FUNCTION_BLOCK INITswitch
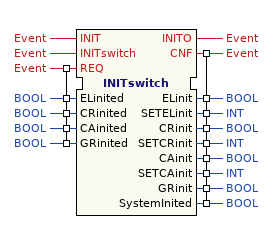
  EVENT_INPUT
    INIT;
    INITswitch;
    REQ WITH ELinited, CRinited, CAinited, GRinited;
  END_EVENT
  EVENT_OUTPUT
    INITO;
    CNF WITH ELinit, SETELinit, CRinit, SETCRinit, CAinit, SETCAinit, GRinit, SystemInited;
  END_EVENT
  VAR_INPUT
    ELinited : BOOL;
    CRinited : BOOL;
    CAinited : BOOL;
    GRinited : BOOL;
  END_VAR
  VAR_OUTPUT
    ELinit : BOOL;
    SETELinit : INT;
    CRinit : BOOL;
    SETCRinit : INT;
    CAinit : BOOL;
    SETCAinit : INT;
    GRinit : BOOL;
    SystemInited : BOOL;
  END_VAR
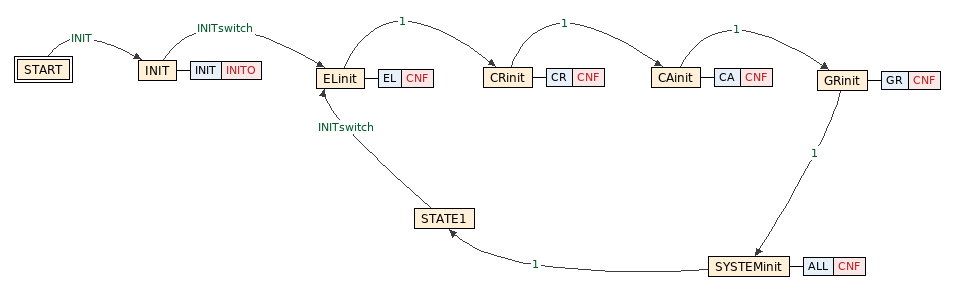
  EC_STATES
    START;
    INIT : INIT -> INITO;
    ELinit : EL -> CNF;
    CRinit : CR -> CNF;
    CAinit : CA -> CNF;
    GRinit : GR -> CNF;
    SYSTEMinit : ALL -> CNF;
    STATE1;
  END_STATES
  EC_TRANSITIONS
    START TO INIT := INIT;
    INIT TO ELinit := INITswitch;
    ELinit TO CRinit := 1;
    CRinit TO CAinit := 1;
    CAinit TO GRinit := 1;
    GRinit TO SYSTEMinit := 1;
    SYSTEMinit TO STATE1 := 1;
    STATE1 TO ELinit := INITswitch;
  END_TRANSITIONS
  ALGORITHM INIT IN ST:
CAinit := FALSE;&#38;#10;CRinit := FALSE;&#38;#10;ELinit := FALSE;&#38;#10;GRinit := FALSE;&#38;#10;SystemInited := FALSE;&#38;#10;
  END_ALGORITHM
  ALGORITHM EL IN ST:
ELinit := TRUE;&#38;#10;SETELinit := 0;&#38;#10;CAinit := FALSE;&#38;#10;CRinit := FALSE;&#38;#10;GRinit := FALSE;&#38;#10;
  END_ALGORITHM
  ALGORITHM CR IN ST:
CRinit := TRUE;&#38;#10;SETCRinit := 0;&#38;#10;CAinit := FALSE;&#38;#10;ELinit := FALSE;&#38;#10;GRinit := FALSE;&#38;#10;
  END_ALGORITHM
  ALGORITHM CA IN ST:
CAinit := TRUE;&#38;#10;SETCAinit := 1;&#38;#10;CRinit := FALSE;&#38;#10;ELinit := FALSE;&#38;#10;GRinit := FALSE;&#38;#10;
  END_ALGORITHM
  ALGORITHM GR IN ST:
GRinit := TRUE;&#38;#10;CAinit := FALSE;&#38;#10;CRinit := FALSE;&#38;#10;ELinit := FALSE;&#38;#10;
  END_ALGORITHM
  ALGORITHM ALL IN ST:
SystemInited := TRUE;&#38;#10;CAinit := FALSE;&#38;#10;CRinit := FALSE;&#38;#10;ELinit := FALSE;&#38;#10;GRinit := FALSE;&#38;#10;
  END_ALGORITHM
END_FUNCTION_BLOCK
